{attribute 'GeneratedUsingTerminal: EL2252--0000'}
{attribute addProperty BoxType "EL2252--0000"}
{attribute addProperty Description "EL2252 2Ch. Dig. Output 24V, 0.5A, DC Time Stamp"}
{attribute addProperty Physics "KK"}
{attribute addProperty Id "DC_Sync_ActivateAT %Q*DC_Sync_Activate_FA2D29101DC_Sync_StartAT %Q*DC_Sync_Start_9CCB0E514Channel_1AT %Q*Channel_42CA91F71Channel_2AT %Q*Channel_42CA91F71WcStateAT %I*WcState_0B2B16F91InfoDataAT %I*InfoData_A7436BC610"}
{attribute addProperty CRC "4287864240"}
{attribute addProperty Size "18"}
TYPE EL2252_FF939DB0 EXTENDS EtcSlaveTerminalBase_947E5A46 :
STRUCT
	{attribute addProperty Name "DC_Sync_Activate"}
	DC_Sync_Activate : DC_Sync_Activate_FA2D2910;
	{attribute addProperty Name "DC_Sync_Start"}
	DC_Sync_Start : DC_Sync_Start_9CCB0E51;
	{attribute addProperty Name "Channel_1"}
	Channel_1 : Channel_42CA91F7;
	{attribute addProperty Name "Channel_2"}
	Channel_2 : Channel_42CA91F7;
	{attribute addProperty Name "WcState"}
	WcState : WcState_0B2B16F9;
	{attribute addProperty Name "InfoData"}
	InfoData : InfoData_A7436BC6;
END_STRUCT
END_TYPE

(* stored: Version 1.2.0.0, ProductVersion 3.1.4024.9
   DUT EL2252_FF939DB0: Id {ebe797a7-9771-40aa-9e40-3bad02ce6d73} *)
